# EPICS autosave request: iocBoot/obsolete/ioc13lab2/auto_settings.req
#file "Keithley2kDMM_mf10_settings.req", P=$(P), Dmm=DMM1
file "scan_settings.req", P=$(P), S=scan1
file "scan_settings.req", P=$(P), S=scan2
file "scan_settings.req", P=$(P), S=scan3
file "scan_settings.req", P=$(P), S=scan4
file "CARS_8_motor_settings.req", P=$(P)
